FUNCTION_BLOCK QualityInspectionSequenceFaultReaction EXTENDS QualityInspectionSequence IMPLEMENTS ZCore.ISequence
VAR
  _step : ZCore.Step(QualityInspectionStep.FaultReactionBegin, QualityInspectionStep.FaultReactionEnd);
  _timerSim : ZAux.Timer;
END_VAR

IF OnStart(_step) THEN
  ; // init custom sequence variables here ...
END_IF

REPEAT
  LogStep();

  CASE _step.Index OF
    (* -------------------------------------------------------------------------------------------------------------------------------- *)
    QualityInspectionStep.FaultReactionBegin:
    (* -------------------------------------------------------------------------------------------------------------------------------- *)
      IF _step.OnEntry()
      THEN
        _timerSim.WaitAsync(5);
			END_IF
      
      Await(_timerSim, nextStep:=QualityInspectionStep.FaultReactionEnd);
      // _step.SetNext(index:=QualityInspectionStep.FaultReactionEnd);

    (* -------------------------------------------------------------------------------------------------------------------------------- *)
    QualityInspectionStep.FaultReactionEnd:
    (* -------------------------------------------------------------------------------------------------------------------------------- *)    
      SetBusy(FALSE);
  
  ELSE
    Abort('sequence contains unhandled step');
  END_CASE
UNTIL _step.IsNotRepeatable() OR_ELSE NOT Busy END_REPEAT

END_FUNCTION_BLOCK

(* stored: Version 1.1.0.1
   POU QualityInspectionSequenceFaultReaction: Id {13dbc3ef-d432-4d1d-94a1-53fa55faa0df}, SpecialFunc None *)
